TYPE ST_Machine_Status :
	STRUCT
		HomeComplete : BOOL;
	END_STRUCT
END_TYPE

(* stored: Version 1.1.0.1
   DUT ST_Machine_Status: Id {1137c440-9402-4f8f-b8f9-11f0b24c29c7} *)
